TYPE MastLightReq :
STRUCT

RedReq: BOOL;
RedFlashReq: BOOL;
YelReq: BOOL;
YelFlashReq: BOOL;
GrnReq: BOOL;
GrnFlashReq: BOOL;
HornReq: BOOL;	

END_STRUCT
END_TYPE

(* stored: Version 1.1.0.1, ProductVersion 3.1.4024.6
   DUT MastLightReq: Id {4022043c-fd1e-4e62-80ab-5719a660e203} *)
